{attribute 'GeneratedUsingTerminal: EK1122-0000-0018'}
{attribute addProperty BoxType "EK1122-0000-0018"}
{attribute addProperty Id "Beckhoff_EL67xxsub_EK1100EK1100_AB5A94672"}
{attribute addProperty CRC "2792157112"}
{attribute addProperty Size "2"}
TYPE Beckhoff_EL67xxEK1122_A66CEFB8 EXTENDS EK1122_AB5A9467 :
STRUCT
	{attribute addProperty Name "Beckhoff_EL67xxsub_EK1100"}
	{attribute addProperty PreviousPort "Beckhoff EL67xxEK1122 : D"}
	Beckhoff_EL67xxsub_EK1100 : EK1100_AB5A9467;
END_STRUCT
END_TYPE

(* stored: Version 1.2.0.0, ProductVersion 3.1.4024.9
   DUT Beckhoff_EL67xxEK1122_A66CEFB8: Id {6c64dd91-e4ad-433f-9bfe-d64703ca48d6} *)
